// TIA Portal V19 export
FUNCTION_BLOCK "UP_Saeure.GP0x"   // FB1002, LAD
TITLE = Pumpe Umwälzpumpe Säure
{ S7_Optimized_Access := 'TRUE' }
// Funktionen: Umwälzen / Entsorgung
// stored: AutoNumber false, MemoryReserve 100, SetENOAutomatically false
   VAR RETAIN
      In { ExternalAccessible := 'False'; ExternalVisible := 'False'; ExternalWritable := 'False'} : Struct
         NotHalt : Bool;
         ext_Freigabe : Bool;   // Kein Gasalarm, Kein Notstrom
         TW_senkt : Bool;
         Auto : Bool;   // Paneltaste
         Ein : Bool;   // Paneltaste
         Quitt_Al_Dfl : Bool;
         FU_betriebsbereit : Bool;
         FU_Stoerung : Bool;
         Niv_TLS : Bool;
         Niv_min : Bool;
         Niv_max : Bool;
         Niv_Uel : Bool;
         Frg_Niv_CM05 : Bool;
         SRM_Saugseite_auf : Bool;
         SRM_Saugseite_zu : Bool;
         SRM_Druckseite_auf : Bool;
         SRM_Druckseite_zu : Bool;
         SRM_Eingang_Spülltg_auf : Bool;
         SRM_Eingang_Spülltg_zu : Bool;
         SRM_Ausgang_Spülltg_auf : Bool;
         SRM_Ausgang_Spülltg_zu : Bool;
         SRM_Entsogung_UV02_auf : Bool;
         SRM_Entsogung_UV02_zu : Bool;
         SRM_UV02_GP01_auf : Bool;
         SRM_UV02_GP01_zu : Bool;
         SRM_UV02_GP02_auf : Bool;
         SRM_UV02_GP02_zu : Bool;
         "SRM_GP02.QM41_auf" : Bool;
         "SRM_GP01.QM14_auf" : Bool;
         Anf_HF_Ents_CM0x : Bool;
         GW_p_UP : Bool;
         GW_LF_UP : Bool;
         Imp_Dfl : Bool;
         GW_Dfl : Bool;
         Tuer_zu_Seite_GP01 : Bool;
         Tuer_zu_vorn_GP01 : Bool;
         Tuer_zu_vorn_GP02 : Bool;
         Leckage_Doppelrohr_ok_BL26 : Bool;
         Leckage_Doppelschlauch_ok_BL33 : Bool;
         Leckage_Uml_Tunnel_ok_BL34 : Bool;
         Leckage_PFA_Uebergang_ok_BL16 : Bool;
         Leckage_PFA_Uebergang_ok_BL25 : Bool;
         Betriebsart : USInt := 0;   // Paneltaste
         FU_speed : Int;
         Druck_Pumpe : Real;
      END_STRUCT;
      Param { ExternalAccessible := 'False'; ExternalVisible := 'False'; ExternalWritable := 'False'} : Struct
         SW_Hand : Int;   // [%]
         SW_Auto_AZ : Int;   // [%]
         SW_Auto_aAZ : Int;   // [%]
         Spülzeit : Time;
         DT_Druckaufbau : Time;
         DT_Testzeit : Time;
         SW_Drucktest : Real;
         "Name" : String[12];
      END_STRUCT;
      Zst { ExternalAccessible := 'False'; ExternalVisible := 'False'; ExternalWritable := 'False'} : Struct
         Niveau : USInt;
         Status_GP0x : USInt;
         Status_DT : USInt;
         Restzeit_Spülen : Time;
         Restzeit_DT : Time;
         Spuelen : Bool;
         Spuelen_aktiv : Bool;
         Drucktest_aktiv : Bool;
         Umwaelzen : Bool;
         Weg_frei : Bool;
         Zeit_laeuft : Bool;
         Drucktest_ok : Bool;
         Bedienung_erlaubt : Bool;
         speed : Int;   // [%]
      END_STRUCT;
      Mld { ExternalAccessible := 'False'; ExternalVisible := 'False'; ExternalWritable := 'False'} : Struct
         Niv_TLS : Bool;
         Niv_Ueberlauf : Bool;
         Niv_Sensorfehler : Bool;
         GW_p_UP : Bool;
         GW_LF_UP : Bool;
         GW_Dfl : Bool;
         UeW_Dfl_Ents : Bool;
         FU_nicht_bereit : Bool;
         FU_Stoerung : Bool;
         n_Auto : Bool;
         TO_Druckaufbau : Bool;
         Drucktest_ok : Bool;
         DT_Fehler : Bool;
         Pu_Spuelen_Fertig : Bool;
      END_STRUCT;
      Out { ExternalAccessible := 'False'; ExternalVisible := 'False'; ExternalWritable := 'False'} : Struct
         GP0x_Ein : Bool;
         Ventil_Saugseite : Bool;
         Ventil_Druckseite : Bool;
         Spülventil_Eingang : Bool;
         Spülventil_Ausgang : Bool;
         Entsorgung_UV02 : Bool;
         Ventil_UV02_GP01 : Bool;
         Ventil_UV02_GP02 : Bool;
         Soll_speed : Int;
      END_STRUCT;
   END_VAR
   VAR
      IEC_Timer { ExternalAccessible := 'False'; ExternalVisible := 'False'; ExternalWritable := 'False'} : Struct
         Spülen { S7_SetPoint := 'True'} : TP_TIME;
         GW_p { S7_SetPoint := 'True'} : TON_TIME;
         GW_Dfl { S7_SetPoint := 'True'} : TON_TIME;
         Imp_Dfl { S7_SetPoint := 'True'} : TON_TIME;
         Drucktest { S7_SetPoint := 'True'} : TP_TIME;
         TO_Druckaufbau { S7_SetPoint := 'True'} : TON_TIME;
         Spülventil_Ausgang { S7_SetPoint := 'True'} : TOF_TIME;
      END_STRUCT;
      R_TRIG_Hand_EIN { ExternalAccessible := 'False'; ExternalVisible := 'False'; ExternalWritable := 'False'} : R_TRIG;
   END_VAR
   VAR_TEMP
      Spülzeit : Time;
      Zeit_DT : Time;
      posFl_Hand : Bool;
      Leckage_Entsorgung_ok_GP01 : Bool;
      Leckage_Entsorgung_ok_GP02 : Bool;
      Alarm_Dfl_Ents : Bool;
   END_VAR
   VAR CONSTANT
      Niv_TLS : USInt := 7;
      Niv_Min : USInt := 70;
      Niv_max : USInt := 85;
      Niv_Uel : USInt := 98;
      S1 : USInt := 1;
      S2 : USInt := 2;
      S3 : USInt := 3;
      S4 : USInt := 4;
   END_VAR
BEGIN

REGION Network 1 (SCL): Input
   // Panelbedienung und Sensoren --> Input()
   // Not-Halt
   #In.NotHalt := NOT "DB_PNOZ_IN_Out".In.NH_Frg_Pumpen OR NOT "E_Frg_AbLW";

    // positive Flanke "Hand Ein"
   #R_TRIG_Hand_EIN(CLK := #In.Ein,
                    Q => #posFl_Hand);

   // Leckage Entsorgung
   #Leckage_Entsorgung_ok_GP01 :=#In.Leckage_PFA_Uebergang_ok_BL16 AND #In.Leckage_Doppelrohr_ok_BL26 AND #In.Leckage_Uml_Tunnel_ok_BL34;

   #Leckage_Entsorgung_ok_GP02 := #In.Leckage_PFA_Uebergang_ok_BL25 AND #In.Leckage_Doppelrohr_ok_BL26 AND #In.Leckage_Doppelschlauch_ok_BL33;

   // Quittierung Alarm Durchfluss
   IF #In.Quitt_Al_Dfl AND #Mld.UeW_Dfl_Ents THEN
       #Mld.UeW_Dfl_Ents := FALSE;
   END_IF;
END_REGION

REGION Network 2 (SCL): Ansteuerung
   // Alles AUS
   IF (#In.Betriebsart = 3) AND #In.ext_Freigabe THEN // Spülen
       #IEC_Timer.Spülventil_Ausgang(IN := #Out.Spülventil_Eingang,
                                     PT := T#3s,
                                     Q => #Out.Spülventil_Ausgang);
   ELSE
       #Out.Spülventil_Eingang := FALSE;
       #Out.Spülventil_Ausgang := FALSE;
   END_IF;
   #Zst.Restzeit_Spülen := T#0s;
   #Out.Ventil_Saugseite := FALSE;
   #Out.Ventil_Druckseite := FALSE;
   #Out.Entsorgung_UV02 := FALSE;
   #Out.Ventil_UV02_GP01 := FALSE;
   #Out.Ventil_UV02_GP02 := FALSE;

   // "Normal"-Betrieb
   #Zst.Bedienung_erlaubt := NOT #In.Ein AND NOT #In.Auto AND NOT #Mld.DT_Fehler;

   //Drucktest rücksetzen
   IF #In.Betriebsart <> 4 OR #Zst.Spuelen_aktiv OR #Zst.Umwaelzen OR NOT #In.Ein THEN
       #Mld.Drucktest_ok := FALSE;
       // #Mld.DT_Fehler := FALSE;
       #Mld.TO_Druckaufbau := FALSE;
       #Zst.Status_DT := 0;
       #Zst.Drucktest_aktiv := FALSE;
   END_IF;
   //Spülmeldung rücksetzen
   IF #In.Betriebsart <> 3 OR NOT #In.Ein THEN
       #Mld.Pu_Spuelen_Fertig := FALSE;
   END_IF;

   IF #In.ext_Freigabe THEN
       CASE #In.Betriebsart OF
           0:  // Umwälzen
                     // Ventile öffnen
               #Out.Ventil_Saugseite := (#In.Auto OR #In.Ein) AND #In.Niv_TLS AND NOT #In.TW_senkt
               AND #In.SRM_Ausgang_Spülltg_zu AND #In.SRM_Eingang_Spülltg_zu;
               #Out.Ventil_Druckseite := #Out.Ventil_Saugseite AND NOT #In.Anf_HF_Ents_CM0x;

               // Verwerfen Auto
               #Out.Ventil_UV02_GP01 := #In.Anf_HF_Ents_CM0x AND #In."SRM_GP01.QM14_auf" AND #In.Auto
               AND #In.Tuer_zu_Seite_GP01 AND #In.Tuer_zu_vorn_GP01 AND #Leckage_Entsorgung_ok_GP01;

               #Out.Ventil_UV02_GP02 := #In.Anf_HF_Ents_CM0x AND #In."SRM_GP02.QM41_auf" AND #In.Auto
               AND #In.Tuer_zu_vorn_GP02 AND #Leckage_Entsorgung_ok_GP02;

               // Check Weg Verwerfen
               #Zst.Weg_frei := #In.SRM_Saugseite_auf AND
               (#In.SRM_UV02_GP01_auf AND #In.SRM_UV02_GP02_zu OR
               #In.SRM_UV02_GP02_auf AND #In.SRM_UV02_GP01_zu);

               #Out.Entsorgung_UV02 := #In.Anf_HF_Ents_CM0x AND #Zst.Weg_frei AND NOT #Mld.UeW_Dfl_Ents;

               // Wenn geöffnet --> Frg Pumpe
               #Zst.Umwaelzen := (#In.SRM_Druckseite_auf AND  #In.SRM_Saugseite_auf) OR  (#Zst.Weg_frei AND #In.SRM_Entsogung_UV02_auf) ;

           1:  // Entsorgung --> GP02
                         // Ventile öffnen
               #Out.Ventil_Saugseite := #In.Ein AND #In.Niv_TLS AND #In.SRM_Ausgang_Spülltg_zu AND #In.SRM_Eingang_Spülltg_zu;
               #Out.Ventil_Druckseite := FALSE;

               // Verwerfen 
               #Out.Ventil_UV02_GP02 := #In.Ein AND #In."SRM_GP02.QM41_auf" AND #In.Tuer_zu_vorn_GP02
               AND #Leckage_Entsorgung_ok_GP02;

               // Check Weg Verwerfen
               #Zst.Weg_frei := #In.SRM_Saugseite_auf AND #In.SRM_UV02_GP02_auf AND #In.SRM_UV02_GP01_zu;

               #Out.Entsorgung_UV02 := #In.Ein AND #Zst.Weg_frei;

               // Wenn geöffnet --> Frg Pumpe
               #Zst.Umwaelzen := #Zst.Weg_frei AND #In.SRM_Entsogung_UV02_auf;

           2:  // Entsorgung --> GP01
                        // Ventile öffnen
               #Out.Ventil_Saugseite := #In.Ein AND #In.Niv_TLS AND #In.SRM_Ausgang_Spülltg_zu AND #In.SRM_Eingang_Spülltg_zu;
               #Out.Ventil_Druckseite := FALSE;

               // Verwerfen 
               #Out.Ventil_UV02_GP01 := #In.Ein AND #In."SRM_GP01.QM14_auf" AND #In.Tuer_zu_Seite_GP01 AND #In.Tuer_zu_vorn_GP01
               AND #Leckage_Entsorgung_ok_GP01;

               // Check Weg Verwerfen
               #Zst.Weg_frei := #In.SRM_Saugseite_auf AND #In.SRM_UV02_GP01_auf AND #In.SRM_UV02_GP02_zu;

               #Out.Entsorgung_UV02 := #In.Ein AND #Zst.Weg_frei;

               // Wenn geöffnet --> Frg Pumpe
               #Zst.Umwaelzen := #Zst.Weg_frei AND #In.SRM_Entsogung_UV02_auf;

           3: // Spülen - nur Hand
               #Zst.Umwaelzen := FALSE;
               #Zst.Weg_frei := FALSE;

               IF #In.Ein AND #In.Frg_Niv_CM05 THEN
                       IF #posFl_Hand THEN
                           #Zst.Spuelen_aktiv := TRUE;
                       END_IF;
                       #Out.Spülventil_Eingang := #In.SRM_Druckseite_zu AND #In.SRM_Saugseite_zu AND #Zst.Spuelen_aktiv;

                       #IEC_Timer.Spülen(IN := #In.SRM_Eingang_Spülltg_auf AND #In.SRM_Ausgang_Spülltg_auf,
                                         PT := #Param.Spülzeit,
                                         Q => #Zst.Spuelen,
                                         ET => #Spülzeit);
                       #Zst.Restzeit_Spülen := #Param.Spülzeit - #Spülzeit;

                       IF #In.SRM_Eingang_Spülltg_auf AND #In.SRM_Ausgang_Spülltg_auf AND NOT #Zst.Spuelen THEN
                           #Zst.Spuelen_aktiv := FALSE;
                           #Out.Spülventil_Eingang := FALSE;
                       END_IF;

                       // Fertig
                       IF NOT #Zst.Spuelen AND NOT #Zst.Spuelen_aktiv AND NOT #Out.Spülventil_Ausgang THEN
                           #Out.Spülventil_Eingang := FALSE;
                           #Out.Spülventil_Ausgang := FALSE;
                           #Zst.Restzeit_Spülen := T#0s;
                           #Mld.Pu_Spuelen_Fertig := TRUE;
                       END_IF;
                   ELSE
                       #Zst.Spuelen := FALSE;
                       #Out.Spülventil_Eingang := FALSE;
                       #Out.Spülventil_Ausgang := FALSE;
                       #Zst.Restzeit_Spülen := T#0s;
                   END_IF;

           4: // Spülen + Drucktest - nur Hand
               #Zst.Umwaelzen := FALSE;
               #Zst.Weg_frei := FALSE;
            IF NOT #Zst.Drucktest_aktiv THEN
                   IF #In.Ein AND #In.Frg_Niv_CM05 THEN
                       IF #posFl_Hand THEN
                           #Zst.Spuelen_aktiv := TRUE;
                       END_IF;
                       #Out.Spülventil_Eingang := #In.SRM_Druckseite_zu AND #In.SRM_Saugseite_zu;
                       #Out.Spülventil_Ausgang := #Out.Spülventil_Eingang;

                       #IEC_Timer.Spülen(IN := #In.SRM_Eingang_Spülltg_auf AND #In.SRM_Ausgang_Spülltg_auf,
                                         PT := #Param.Spülzeit,
                                         Q => #Zst.Spuelen,
                                         ET => #Spülzeit);
                       #Zst.Restzeit_Spülen := #Param.Spülzeit - #Spülzeit;

                       IF #In.SRM_Eingang_Spülltg_auf AND #In.SRM_Ausgang_Spülltg_auf AND NOT #Zst.Spuelen THEN
                           #Zst.Spuelen_aktiv := FALSE;
                       END_IF;

                       // Fertig
                       IF NOT #Zst.Spuelen AND NOT #Zst.Spuelen_aktiv THEN
                           #Out.Spülventil_Eingang := FALSE;
                           #Out.Spülventil_Ausgang := FALSE;
                           #Zst.Restzeit_Spülen := T#0s;
                            #Zst.Drucktest_aktiv := TRUE;
                            #Zst.Status_DT := #S1;
                       END_IF;
                   ELSE
                       #Zst.Spuelen := FALSE;
                       #Out.Spülventil_Eingang := FALSE;
                       #Out.Spülventil_Ausgang := FALSE;
                       #Zst.Restzeit_Spülen := T#0s;
                   END_IF;
                END_IF;

                IF #Zst.Drucktest_aktiv THEN

                    CASE #Zst.Status_DT OF

                        #S1:  //Druckaufbau
                            IF "DB_Temporaer".Drucksensoren_deaktiviert THEN//20.01.22
                                #Zst.Drucktest_ok := TRUE;

                                "Ergebnis_DT"("Name" := #Param.Name,
                                              akt_Zeit := "Uhrzeit".aktDatum,
                                              ok := #Zst.Drucktest_ok,
                                              Fehler := NOT #Zst.Drucktest_ok);

                                #Mld.Drucktest_ok := #Zst.Drucktest_ok;
                                #Mld.DT_Fehler := NOT #Zst.Drucktest_ok;

                                #Zst.Status_DT := #S4;
                            ELSE

                                #Out.Spülventil_Eingang := #In.SRM_Druckseite_zu AND #In.SRM_Saugseite_zu;
                                #Out.Spülventil_Ausgang := FALSE;
                                IF (#In.Druck_Pumpe > #Param.SW_Drucktest + 0.25) OR #Mld.TO_Druckaufbau THEN
                                    #Out.Spülventil_Eingang := FALSE;
                                    #Zst.Status_DT := #S2;
                                END_IF;
                                #Zst.Restzeit_DT := #Param.DT_Druckaufbau - #IEC_Timer.TO_Druckaufbau.ET;
                            END_IF;

                        #S2: //Wartezeit
                           #IEC_Timer.Drucktest(IN := #In.SRM_Eingang_Spülltg_zu,
                                                PT := #Param.DT_Testzeit,
                                                Q => #Zst.Zeit_laeuft,
                                                ET => #Zeit_DT);
                           #Zst.Restzeit_DT := #Param.DT_Testzeit - #Zeit_DT;

                           IF NOT #Zst.Zeit_laeuft AND #In.SRM_Eingang_Spülltg_zu THEN
                               #Zst.Restzeit_DT := T#0s;
                               #Zst.Status_DT := #S3;
                           END_IF;

                       #S3:// Überprüfung
                           #Zst.Drucktest_ok := #In.Druck_Pumpe >= #Param.SW_Drucktest;

                           "Ergebnis_DT"("Name" := #Param.Name,
                                         akt_Zeit := "Uhrzeit".aktDatum,
                                         ok := #Zst.Drucktest_ok,
                                         Fehler := NOT #Zst.Drucktest_ok);

                           #Mld.Drucktest_ok := #Zst.Drucktest_ok;
                           #Mld.DT_Fehler := NOT #Zst.Drucktest_ok;

                           #Zst.Status_DT := #S4;

                       #S4: // Ende
                           ;
                   END_CASE;
               END_IF;
       END_CASE;
   END_IF;

       // Pumpe an    
   #Out.GP0x_Ein := (#Zst.Umwaelzen (*OR #Zst.Spuelen*)) AND NOT #In.NotHalt AND #In.ext_Freigabe;

       // Geschwindigkeitsvorgabe
       // SEW: 100% == 3000 U/min == 15000 Digits
       IF #Out.GP0x_Ein THEN
           IF #In.Ein THEN
               #Out.Soll_speed := #Param.SW_Hand * 150;
           ELSE
               IF "Uhrzeit".AZ_aktiv THEN
                   #Out.Soll_speed := #Param.SW_Auto_AZ * 150;
               ELSE
                   #Out.Soll_speed := #Param.SW_Auto_aAZ * 150;
               END_IF;
           END_IF;
       ELSE
           #Out.Soll_speed := 0;
       END_IF;
END_REGION

REGION Network 3 (SCL): Überwachung / Meldungen
   // Trockenlaufschutz
   #Mld.Niv_TLS := NOT #In.Niv_TLS;
   // Überlauf
   #Mld.Niv_Ueberlauf := #In.Niv_Uel;

   // Durchflussüberwachung
   #IEC_Timer.Imp_Dfl(IN := NOT #In.Imp_Dfl AND #Zst.Umwaelzen AND #Out.Entsorgung_UV02,
                      PT := T#5s,
                      Q => #Alarm_Dfl_Ents);

   IF #Alarm_Dfl_Ents THEN
       #Mld.UeW_Dfl_Ents := TRUE;
   END_IF;

   // Zeitüberschreitung Druckaufbau
   #IEC_Timer.TO_Druckaufbau(IN := #Zst.Status_DT = #S1,
                             PT := #Param.DT_Druckaufbau,
                             Q => #Mld.TO_Druckaufbau);

   // Grenzwert Druck
   #IEC_Timer.GW_p(IN :=#Out.GP0x_Ein AND #In.GW_p_UP,
                   PT := T#3s,
                   Q => #Mld.GW_p_UP);

   #IEC_Timer.GW_Dfl(IN := #In.GW_Dfl AND #Out.GP0x_Ein AND #In.SRM_Druckseite_auf AND #Out.Entsorgung_UV02,
                     PT := T#15s,
                     Q => #Mld.GW_Dfl);

   // Grenzwert Leitfähigkeit Düsen Umwälzung
   #Mld.GW_LF_UP := #In.GW_LF_UP;

   // Frequenzumrichter 24V-Betrieb
   #Mld.FU_nicht_bereit := NOT #In.FU_betriebsbereit AND NOT #In.NotHalt;
   // Störung Frequenzumrichter
   #Mld.FU_Stoerung := #In.FU_Stoerung AND NOT #In.NotHalt;
   // nicht in Automatik
   #Mld.n_Auto := NOT #In.Auto AND "DB_ANLAGE".BA.Automat_ein;
END_REGION

REGION Network 4 (SCL): --> Visu
   // Status Pumpe
   "Status_E0A"(Hand := #In.Ein,
                Auto := #In.Auto,
                SonderModus_PumpeSpuelen:=#Zst.Spuelen,
                Stoerung := #In.FU_Stoerung OR NOT #In.FU_betriebsbereit,
                Ausgang := #Out.GP0x_Ein,
                StatusByte => #Zst.Status_GP0x);

   // Ist-Geschwindigkeit FU
   // SEW: 100% == 3000 U/min == 15000 Digits
   #Zst.speed := #In.FU_speed / 150; // in[%]

   // Anzeige Füllstand
   "Niv_Visu"(Niv_1 := #In.Niv_TLS,
              Niv_2 := #In.Niv_min,
              Niv_3 := #In.Niv_max,
              Niv_4 := #In.Niv_Uel,
              Niv_5 := FALSE,
              Niv_6 := FALSE,
              Wert_1 := #Niv_TLS,
              Wert_2 := #Niv_Min,
              Wert_3 := #Niv_max,
              Wert_4 := #Niv_Uel,
              Wert_5 := 0,
              Wert_6 := 0,
              Niveau => #Zst.Niveau,
              Niv_Err => #Mld.Niv_Sensorfehler);
END_REGION
END_FUNCTION_BLOCK
